FUNCTION_BLOCK ContactorReverse
VAR
	_output AT%QX1.1: BOOL;
END_VAR

PROPERTY State : BOOL
GET
State := _output;
END_GET
SET
_output := State;
END_SET
END_PROPERTY

END_FUNCTION_BLOCK

(* stored: Version 1.1.0.1, ProductVersion 3.1.4024.12
   POU ContactorReverse: Id {cbb906b0-fc51-40c3-90e9-12890d021e59}, SpecialFunc None
   Property State: Id {071cc637-4931-422d-8ca2-244b0a22f730}
   Get Get: Id {770dd012-0daa-4b75-84bd-579a6dc1884e}
   Set Set: Id {f37c17f1-7c1f-4962-bb94-35c1514b4e44} *)
